// Mitsubishi GX Works2 project: ZhaoQing_OCV_1_9   PLC: Q06UDEH

TYPE ConveyorIO : STRUCT
  xCWPresent : BOOL;  (* 正转检测有无传感器 *)
  xCCWPresent : BOOL;  (* 反转检测有无传感器 *)
  xLoad : BOOL;  (* 上料请求 *)
  xUnload : BOOL;  (* 下料请求 *)
  xMotorCW : BOOL;  (* 电机正转 *)
  xMotorCCW : BOOL;  (* 电机反转 *)
  xEmpty : BOOL;  (* 线体状态为空 *)
  xNextRun : BOOL;  (* 下段线体运行 *)
  xUnloadCCW : BOOL;  (* 下料为反转 *)
  xloadCCW : BOOL;  (* 上料为反转 *)
  xForward : BOOL;  (* 正转手动 *)
  xBackward : BOOL;  (* 反转手动 *)
  xBusy : BOOL;  (* 工作中 *)
  xPutInto : BOOL;  (* 线体直接投入物料 *)
  xLoadAlarrm : BOOL;  (* 上料报警 *)
  xUnloadAlarm : BOOL;  (* 下料报警 *)
  iProductCategory : INT;  (* 产品种类 *)
  tLoadDelay : TIME;  (* 进入延时设置 *)
  tUnloadAlarmDelay : TIME;  (* 下料时间设置 *)
  xNotArriveAlarm : BOOL;  (* 未到达报警 *)
END_STRUCT END_TYPE

TYPE ShuttleCarIO : STRUCT
  xReady : BOOL;  (* 准备就绪 *)
  xForward : BOOL;  (* 正转 *)
  xBackward : BOOL;  (* 反转 *)
  iCurrentPos : INT;  (* 当前位置 *)
  iDestinationPos : INT;  (* 目标位置 *)
  xCW : BOOL;  (* 正转输出 *)
  xCCW : BOOL;  (* 反转输出 *)
  xBrake : BOOL;  (* 刹车 *)
  xHomeSwitch : BOOL;  (* 零位接近开关 *)
  xPosLimit : BOOL;  (* 正限位 *)
  xNegLimit : BOOL;  (* 负限位 *)
  xMDIExe : BOOL;  (* MDI开始 *)
  xMDIDone : BOOL;  (* MDI 完成 *)
  xPassLimit : BOOL;  (* 限位屏蔽 *)
  xPosLimitCatch : BOOL;  (* 正限位捕捉 *)
  xNegLimitCatch : BOOL;  (* 负限位捕捉 *)
  xHomeExe : BOOL;  (* 开始寻零 *)
  xHomeDone : BOOL;  (* 寻零完成 *)
  xHomeBusy : BOOL;  (* 寻零中 *)
  xHomeFailed : BOOL;  (* 寻零失败 *)
  xBusy : BOOL;  (* 工作中 *)
END_STRUCT END_TYPE

TYPE SwitchIO : STRUCT
  xLiftCylinderRetractDetect : BOOL;
  xLiftCylinderExtendDetect : BOOL;
  xLiftCylinderRetract : BOOL;
  xLiftCylinderExtend : BOOL;
  xEntryBarCylinderRetract : BOOL;
  xLiftCylinderExtendInit : BOOL;
  xEntryEnable : BOOL;
  xExitEnable : BOOL;
  xExitBarCylinderRetract : BOOL;
  xSwithEnable : BOOL;
  xLiftCylinderRetractButton : BOOL;
  xLiftCylinderExtendButton : BOOL;
  xEntryBarCylinderRetractButton : BOOL;
  xExitBarCylinderRetractButton : BOOL;
END_STRUCT END_TYPE

TYPE BarCylinderIO : STRUCT
  xBarCylinderButton : BOOL;  (* 阻挡气缸 *)
  xPresentSwitch : BOOL;  (* 行程开关 *)
  xBarCylinder : BOOL;  (* 阻挡气缸 *)
  xLoad : BOOL;  (* 上料 *)
  xEmpty : BOOL;  (* 为空指示 *)
  xNextRun : BOOL;  (* 下位设备开始运行 *)
  xUnload : BOOL;  (* 下料 *)
  xTransportMotorCWButton : BOOL;  (* 输送电机正转按钮 *)
  xTransportMotorCW : BOOL;  (* 输送电机正转 *)
  xTransportMotorCCWButton : BOOL;  (* 输送电机反转按钮 *)
  xTransportMotorCCW : BOOL;  (* 输送电机反转 *)
  iProductCategory : INT;  (* 产品种类 *)
  tLoadDelay : TIME;  (* 上料延时 *)
END_STRUCT END_TYPE

// global labels: Global1
VAR_GLOBAL
  g_xAuto AT M11 : BOOL;
  g_xManual : BOOL;
  g_xEStop AT X0BC : BOOL;
  g_xReset AT X0BE : BOOL;
  g_xStackLampRed AT Y2C1 : BOOL;
  g_xStackLampAmber AT Y2C3 : BOOL;
  g_xStackLampGreen AT Y2C2 : BOOL;
  g_xBuzzer AT Y2C4 : BOOL;
  g_xStop AT M2 : BOOL;
  g_xLocalAutoStart AT M1 : BOOL;
  g_xRemoteAutoStart AT M0 : BOOL;
  g_xRemoteAuto AT M10 : BOOL;
  g_iState AT D40 : INT;
  g_iLocalAutoStep : BOOL;
  g_xAlarm : BOOL;
END_VAR

// task Task_01 (event TRUE, interval 0, priority 31): POU, Start

FUNCTION_BLOCK Conveyor
VAR
  m_tLoadTimer : TIME;  (* 上料延时 *)
  m_tonNotArriveAlarm : TON;  (* 未到达报警计时 *)
  m_tonUnloadAlam : TON;  (* 下料报警定时器 *)
  m_tonLoadDelay : TON;  (* 上料延时 *)
  m_tUnloadTimer : TIME;  (* 下料计时器 *)
  iStep : INT;  (* 上料步骤 *)
  m_tNotArriveCurrentTime : TIME;  (* 未到达报警计时当前时间 *)
  m_xInitial : BOOL;  (* 初始化 *)
  m_xLoadDelayOut : BOOL;  (* 上料延时输出 *)
END_VAR
VAR_IN_OUT
  ConveyorMotor : ConveyorIO;  (* 输送线输入输出 *)
END_VAR
(*////////////////////////////////////////////////////////////////////////////////////////////////////////////
//传输线控制FB块，可控制单方向线体，双向旋转线体，支持双向上下料            
//线体初始化后为空的情况下输入xLoad信号即可进行上料动作，使用xLoadCCW信号可反方向上料
//增加了产品信息和产品种类的储存，当传输线为空和上料进行标志位为零的情况下清除产品信息和产品种类
//使用方式是在置位xLoad信号后，把产品信息和产品种类传入，等下料后自动清零
//线体不为空的情况下使用xUnload信号可进行下料动作，物料有无传感器的下降沿后出发计时器，延时断开传输线旋转
//单方向传输线体把xLoadCCW、xUnloadCCW设置为零，双向线体上料方向和下料反向的,方向固定的 把xUnloadCCW设置为1
//双方向线体双向都能上下料的要根据上料的方向来设置xLoadCCW,xUnloadCCW
//增加工作中信号xBusy当电机正转 显示为工作中
//增加上下料超时报警，xLoadAlarm，xUnloadAlarm，设定时间在LOAD_UNLOAD_TIME常量上，现在设置的为30秒
//增加xPutInto信号，用于直接投入的物料，检测开关感应到后，直接进入下料流程，上升沿有效
//离开延时改为变量 iLeaveDelay 默认为0 离开检测开关离输送线尾端比较远的线体需要根据情况设定100ms为单位
增加初始化标志位，增加进入延时时间，初始化为进入延时时间为0 ，离开延时时间为2S，通过外围接口可以更改
//修改信息  修改后请增加版本
12-17进行了优化，增加了未到达报警，当物料未传送到下一设备，就报未到达报警，使用xNextRun标志位制作，没有正常到达
第0步，不能跳转到第一步把标志位复位，即出现中断情况，2秒后报警 有问题

//YAO      V1.0
///////////////////////////////////////////////////////////////////////////////////////////////////////////
********************************************************)
IF NOT m_xInitial THEN
	ConveyorMotor.tLoadDelay:=T#0s;
	ConveyorMotor.tUnloadAlarmDelay:=T#30s;
	m_xInitial:=1;
END_IF;               (*初始化设置延时时间*)

CASE iStep OF
	0:
	ConveyorMotor.xMotorCW:=0;
	ConveyorMotor.xMotorCCW:=0;
    IF g_xAuto THEN          (*自动才进下一步*)
		IF (ConveyorMotor.xCWPresent OR ConveyorMotor.xCCWPresent)  THEN
			iStep:=3;
			ConveyorMotor.xEmpty:=0;(*检测到东西去3，复位empty*)
			ELSE
			iStep:=1;
			ConveyorMotor.xEmpty:=1;         (*没东西去1，置位empty*)
		END_IF;
	END_IF;
	1: 
	ConveyorMotor.xNextRun:=0;          (*复位NextRun*)
	IF ConveyorMotor.xLoad AND ConveyorMotor.xEmpty THEN	(*一般load接上一段的NextRun*)
		iStep:=2;                                             (*empty且有进料信号*)
	END_IF;
	2: 
	IF ConveyorMotor.xloadCCW THEN       (*如果正转为上料，则正转*)
		ConveyorMotor.xMotorCCW:=1; 
		ConveyorMotor.xMotorCW:=0;
	ELSE
	    ConveyorMotor.xMotorCW:=1;                (*反转为上料，则反转*)
		ConveyorMotor.xMotorCCW:=0;
	END_IF;
		m_tonLoadDelay(IN:= (ConveyorMotor.xCWPresent AND NOT ConveyorMotor.xloadCCW) 
		                                        OR (ConveyorMotor.xCCWPresent AND ConveyorMotor.xloadCCW) ,
		                               PT:= ConveyorMotor.tLoadDelay ,
		                               Q:= m_xLoadDelayOut ,
		                               ET:= m_tLoadTimer );
	    IF m_xLoadDelayOut THEN 	 
		    iStep:=3;                                             (*相应光电检测到东西，则去3*)
		END_IF;
	3:
	ConveyorMotor.xMotorCW:=0;
	ConveyorMotor.xMotorCCW:=0;
	ConveyorMotor.xEmpty:=0;          (*停转，且复位Empty，表示有料*)
	IF ConveyorMotor.xUnload THEN        (*停止运转，有Unload信号，则去4*)
		 iStep:=4;
	END_IF;
	4:	
	IF ConveyorMotor.xUnloadCCW THEN   (*正转为下料，则正转*)
		ConveyorMotor.xMotorCCW:=1;  
		ConveyorMotor.xMotorCW:=0;
		ELSE
	    ConveyorMotor.xMotorCW:=1;               (*反转为下料，则反转*)
		ConveyorMotor.xMotorCCW:=0;
	END_IF;
	ConveyorMotor.xNextRun:=1;         (*置位NextRun*)
	IF NOT ConveyorMotor.xUnload THEN       (*Unload信号为0则去0*)(*一般Unload由下段的Empty控制，即下段有料，流程走完*)
		istep:=0;
	END_IF;
END_CASE;
IF LDP(TRUE,ConveyorMotor.xPutInto) THEN
	iStep:=0;
END_IF;

(*IF ConveyorMotor.xEmpty AND iStep<>2 THEN
	ConveyorMotor.iProductCategory:=0;
END_IF;*)
IF g_xEStop=0 OR g_xReset THEN
	iStep:=0;
END_IF;	
IF g_xReset THEN
	ConveyorMotor.xNextRun:=0; 
END_IF;
IF g_xManual THEN
	iStep:=0;
	IF ConveyorMotor.xForward 
		AND ConveyorMotor.xBackward=0 
		AND ConveyorMotor.xMotorCCW=0
		AND g_xEStop THEN
		ConveyorMotor.xMotorCW:=1;
		ConveyorMotor.xMotorCCW:=0;
		ELSE
		ConveyorMotor.xMotorCW:=0;
	END_IF;

	IF ConveyorMotor.xBackward 
		AND ConveyorMotor.xForward=0 
		AND ConveyorMotor.xMotorCW=0
		AND g_xEStop  THEN
		ConveyorMotor.xMotorCCW:=1;
		conveyormotor.xMotorCW:=0;
		ELSE
		ConveyorMotor.xMotorCCW:=0;
	END_IF;
END_IF;
IF ConveyorMotor.xMotorCCW        
	OR ConveyorMotor.xMotorCW THEN  
	ConveyorMotor.xBusy:=1;
	ELSE
	ConveyorMotor.xBusy:=0;
END_IF;
m_tonNotArriveAlarm(IN:= iStep=0 AND ConveyorMotor.xNextRun,PT:= T#2s,Q:= ConveyorMotor.xNotArriveAlarm ,ET:= m_tNotArriveCurrentTime );
m_tonUnloadAlam(IN:= iStep=4,PT:=ConveyorMotor.tUnloadAlarmDelay,Q:= ConveyorMotor.xUnloadAlarm,ET:= m_tUnloadTimer );
END_FUNCTION_BLOCK

PROGRAM POU
VAR
  Cylinder12309 : ShuttleCar;
  CylinderIO12309 : ShuttleCarIO;
  ConveyorIO12114 : ConveyorIO;
  Conveyor12114 : Conveyor;
  Conveyor12115 : Conveyor;
  ConveyorIO12115 : ConveyorIO;
  Switch12312 : Switch;
  SwitchIO12312 : SwitchIO;
  Conveyor12123 : Conveyor;
  ConveyorIO12123 : ConveyorIO;
  Conveyor12124 : Conveyor;
  ConveyorIO12124 : ConveyorIO;
  Conveyor12125 : Conveyor;
  ConveyorIO12125 : ConveyorIO;
  Switch12203 : Switch;
  SwitchIO12203 : SwitchIO;
  Conveyor12142 : Conveyor;
  ConveyorIO12142 : ConveyorIO;
  Bar12326 : BarCylinder;
  BarIO12326 : BarCylinderIO;
  Conveyor12116 : Conveyor;
  ConveyorIO12116 : ConveyorIO;
  Cylinder12308 : ShuttleCar;
  CylinderIO12308 : ShuttleCarIO;
  Conveyor12111 : Conveyor;
  ConveyorIO12111 : ConveyorIO;
  Conveyor12112 : Conveyor;
  ConveyorIO12112 : ConveyorIO;
  Switch12311 : Switch;
  SwitchIO12311 : SwitchIO;
  Conveyor12113 : Conveyor;
  ConveyorIO12113 : ConveyorIO;
  Conveyor12120 : Conveyor;
  ConveyorIO12120 : ConveyorIO;
  Conveyor12121 : Conveyor;
  ConveyorIO12121 : ConveyorIO;
  Conveyor12122 : Conveyor;
  ConveyorIO12122 : ConveyorIO;
  Cylinder12307 : ShuttleCar;
  CylinderIO12307 : ShuttleCarIO;
  Conveyor12108 : Conveyor;
  ConveyorIO12108 : ConveyorIO;
  Conveyor12109 : Conveyor;
  ConveyorIO12109 : ConveyorIO;
  Switch12310 : Switch;
  SwitchIO12310 : SwitchIO;
  Conveyor12110 : Conveyor;
  ConveyorIO12110 : ConveyorIO;
  Conveyor12117 : Conveyor;
  ConveyorIO12117 : ConveyorIO;
  Conveyor12118 : Conveyor;
  ConveyorIO12118 : ConveyorIO;
  Conveyor12119 : Conveyor;
  ConveyorIO12119 : ConveyorIO;
  Conveyor12203 : Conveyor;
  ConveyorIO12203 : ConveyorIO;
  Conveyor12143 : Conveyor;
  ConveyorIO12143 : ConveyorIO;
  Switch12330 : Switch;
  ConveyorIO12144 : ConveyorIO;
  SwitchIO12330 : SwitchIO;
  Switch12333 : Switch;  (* OCV2顶升移载 *)
  ConveyorIO12333 : ConveyorIO;  (* OCV2顶升移载进入线体 *)
  ConveyorIO12152 : ConveyorIO;  (* OCV2顶升移载离开线体 *)
  SwitchIO12333 : SwitchIO;  (* OCV2顶升移载 *)
  m_xTS1ExportPermit : BOOL;  (* OCV2顶升移载 *)
  m_xConveyor12114Export : BOOL;  (* 12114线体输出 *)
  ConveyorIO12146 : ConveyorIO;
  m_xTS2ExportPermit : BOOL;
END_VAR
(*1巷道出库线体*)
Cylinder12309(ShuttleCarInOut:=CylinderIO12309);
ShuttleCarCurrentPosition( X43 OR X44 ,X44 ,X43, FALSE, CylinderIO12309.iCurrentPos );
CylinderIO12309.xReady:=TRUE;
CylinderIO12309.xForward:=M30;
CylinderIO12309.xBackward:=M31;
CylinderIO12309.xPosLimit:=1;
CylinderIO12309.xNegLimit:=1;
Y23D:=CylinderIO12309.xCW;
Y23C:=CylinderIO12309.xCCW;

Conveyor12114(ConveyorMotor:=ConveyorIO12114);
ConveyorIO12114.xForward:=M32;
ConveyorIO12114.xCWPresent:=X45;
Y23E:=ConveyorIO12114.xMotorCW;

Conveyor12115(ConveyorMotor:=ConveyorIO12115);
ConveyorIO12115.xForward:=M33;
ConveyorIO12115.xCWPresent:=X46;
Y23F:=ConveyorIO12115.xMotorCW;

Switch12312(ConveyorEntryIO:=ConveyorIO12116 ,
                                                        ConveyorExitIO:=ConveyorIO12123 ,
                                                        SwitchIO:=SwitchIO12312 );
SwitchIO12312.xLiftCylinderExtendButton:=M34;
SwitchIO12312.xLiftCylinderRetractButton:=M35;
Y242:=SwitchIO12312.xLiftCylinderExtend;
Y241:=SwitchIO12312.xLiftCylinderRetract;
SwitchIO12312.xLiftCylinderExtendDetect:=X4B;
SwitchIO12312.xLiftCylinderRetractDetect:=X4C;
ConveyorIO12116.xForward:=M36;
ConveyorIO12116.xCWPresent:=X49 OR X4A;
Y240:=ConveyorIO12116.xMotorCW;
ConveyorIO12123.xForward:=M37;
ConveyorIO12123.xCWPresent:=X49 OR X4A;
Y243:=ConveyorIO12123.xMotorCW;

Conveyor12124(ConveyorMotor:=ConveyorIO12124);
ConveyorIO12124.xForward:=M38;
ConveyorIO12124.xCWPresent:=X4D;
Y244:=conveyorIO12124.xMotorCW;

Conveyor12125(ConveyorMotor:=ConveyorIO12125);
ConveyorIO12125.xForward:=M39;
ConveyorIO12125.xCWPresent:=X4E;
Y245:=conveyorIO12125.xMotorCW;

(*2巷道出库线体*)
Cylinder12308(ShuttleCarInOut:=CylinderIO12308);
ShuttleCarCurrentPosition( X35 OR X36 ,X36 ,X35, FALSE, CylinderIO12308.iCurrentPos );
CylinderIO12308.xReady:=TRUE;
CylinderIO12308.xForward:=M40;
CylinderIO12308.xBackward:=M41;
CylinderIO12308.xPosLimit:=1;
CylinderIO12308.xNegLimit:=1;
Y235:=CylinderIO12308.xCW;
Y236:=CylinderIO12308.xCCW;

Conveyor12111(ConveyorMotor:=ConveyorIO12111);
ConveyorIO12111.xForward:=M42;
ConveyorIO12111.xCWPresent:=X37;
Y237:=ConveyorIO12111.xMotorCW;

Conveyor12112(ConveyorMotor:=ConveyorIO12112);
ConveyorIO12112.xForward:=M43;
ConveyorIO12112.xCWPresent:=X38;
Y238:=ConveyorIO12112.xMotorCW;

Switch12311(ConveyorEntryIO:=ConveyorIO12113 ,
                                                        ConveyorExitIO:=ConveyorIO12120 ,
                                                        SwitchIO:=SwitchIO12311 );
SwitchIO12311.xLiftCylinderExtendButton:=M44;
SwitchIO12311.xLiftCylinderRetractButton:=M45;
Y233:=SwitchIO12311.xLiftCylinderExtend;
Y232:=SwitchIO12311.xLiftCylinderRetract;
SwitchIO12311.xLiftCylinderExtendDetect:=X3D;
SwitchIO12311.xLiftCylinderRetractDetect:=X3E;
ConveyorIO12113.xForward:=M46;
ConveyorIO12113.xCWPresent:=X3B OR X3C;
Y239:=ConveyorIO12113.xMotorCW;
ConveyorIO12120.xForward:=M47;
ConveyorIO12120.xCWPresent:=X3B OR X3C;
Y234:=ConveyorIO12120.xMotorCW;

Conveyor12121(ConveyorMotor:=ConveyorIO12121);
ConveyorIO12121.xForward:=M48;
ConveyorIO12121.xCWPresent:=X3F;
Y23A:=conveyorIO12121.xMotorCW;

Conveyor12122(ConveyorMotor:=ConveyorIO12122);
ConveyorIO12122.xForward:=M49;
ConveyorIO12122.xCWPresent:=X40;
Y23B:=conveyorIO12122.xMotorCW;

(*3巷道出库线体*)
Cylinder12307(ShuttleCarInOut:=CylinderIO12307);
ShuttleCarCurrentPosition( X27 OR X28 ,X28 ,X27, FALSE, CylinderIO12307.iCurrentPos );
CylinderIO12307.xReady:=TRUE;
CylinderIO12307.xForward:=M50;
CylinderIO12307.xBackward:=M51;
CylinderIO12307.xPosLimit:=1;
CylinderIO12307.xNegLimit:=1;
Y228:=CylinderIO12307.xCW;
Y229:=CylinderIO12307.xCCW;

Conveyor12108(ConveyorMotor:=ConveyorIO12108);
ConveyorIO12108.xForward:=M52;
ConveyorIO12108.xCWPresent:=X26;
Y22A:=ConveyorIO12108.xMotorCW;

Conveyor12109(ConveyorMotor:=ConveyorIO12109);
ConveyorIO12109.xForward:=M53;
ConveyorIO12109.xCWPresent:=X25;
Y22B:=ConveyorIO12109.xMotorCW;

Switch12310(ConveyorEntryIO:=ConveyorIO12110 ,
                                                        ConveyorExitIO:=ConveyorIO12117 ,
                                                        SwitchIO:=SwitchIO12310 );
SwitchIO12310.xLiftCylinderExtendButton:=M54;
SwitchIO12310.xLiftCylinderRetractButton:=M55;
Y22D:=SwitchIO12310.xLiftCylinderExtend;
Y22E:=SwitchIO12310.xLiftCylinderRetract;
SwitchIO12310.xLiftCylinderExtendDetect:=X2D;
SwitchIO12310.xLiftCylinderRetractDetect:=X2E;
ConveyorIO12110.xForward:=M56;
ConveyorIO12110.xCWPresent:=X2F OR X30;
Y22C:=ConveyorIO12110.xMotorCW;
ConveyorIO12117.xForward:=M57;
ConveyorIO12117.xCWPresent:=X2F OR X30;
Y22F:=ConveyorIO12117.xMotorCW;

Conveyor12118(ConveyorMotor:=ConveyorIO12118);
ConveyorIO12118.xForward:=M58;
ConveyorIO12118.xCWPresent:=X31;
Y230:=conveyorIO12118.xMotorCW;

Conveyor12119(ConveyorMotor:=ConveyorIO12119);
ConveyorIO12119.xForward:=M59;
ConveyorIO12119.xCWPresent:=X32;
Y231:=conveyorIO12119.xMotorCW;
(*出库分流顶升移载*)
Switch12203(ConveyorEntryIO:=ConveyorIO12142 ,
                                                        ConveyorExitIO:=ConveyorIO12203 ,
                                                        SwitchIO:=SwitchIO12203);
SwitchIO12203.xLiftCylinderExtendButton:=M60;
SwitchIO12203.xLiftCylinderRetractButton:=M61;
SwitchIO12203.xExitBarCylinderRetractButton:=M64;
Y26B:=SwitchIO12203.xExitBarCylinderRetract;
Y269:=SwitchIO12203.xLiftCylinderExtend;
Y268:=SwitchIO12203.xLiftCylinderRetract;
SwitchIO12203.xLiftCylinderExtendDetect:=X88;
SwitchIO12203.xLiftCylinderRetractDetect:=X89;
ConveyorIO12142.xForward:=M62;
ConveyorIO12142.xCWPresent:=X86;
Y281:=ConveyorIO12142.xMotorCW;
ConveyorIO12142.tLoadDelay:=T#1s;
ConveyorIO12203.xForward:=M63;
ConveyorIO12203.xCWPresent:=X86;
Y26A:=ConveyorIO12203.xMotorCW;
SwitchIO12203.xLiftCylinderExtendInit:=0;

Bar12326(BarCylinderIO:=BarIO12326);
BarIO12326.tLoadDelay:=T#2s;
BarIO12326.xBarCylinderButton:=M64;
BarIO12326.xPresentSwitch:=X94;
BarIO12326.xTransportMotorCWButton:=M65;
Y26E:= BarIO12326.xTransportMotorCW;
Y26C:=BarIO12326.xBarCylinder;

Conveyor12143(ConveyorMotor:=ConveyorIO12143);
ConveyorIO12143.xForward:=M66;
ConveyorIO12143.xCWPresent:=XA2;
Y282:=ConveyorIO12143.xMotorCW;
(*OCV1顶升移载*)
Switch12330(ConveyorEntryIO:=ConveyorIO12144 ,
                                                        ConveyorExitIO:=ConveyorIO12146 ,
                                                        SwitchIO:=SwitchIO12330);
SwitchIO12330.xLiftCylinderExtendButton:=M67;
SwitchIO12330.xLiftCylinderRetractButton:=M68;
SwitchIO12330.xExitBarCylinderRetractButton:=M69;
Y286:=SwitchIO12330.xExitBarCylinderRetract;
Y284:=SwitchIO12330.xLiftCylinderExtend;
Y285:=SwitchIO12330.xLiftCylinderRetract;
SwitchIO12330.xLiftCylinderExtendDetect:=XA5;
SwitchIO12330.xLiftCylinderRetractDetect:=XA6;
ConveyorIO12144.xForward:=M70;
ConveyorIO12144.xCWPresent:=XA7;
Y283:=ConveyorIO12144.xMotorCW;
ConveyorIO12146.xForward:=M71;
ConveyorIO12146.xCWPresent:=XA7;
Y280:=ConveyorIO12146.xMotorCW;

(*OCV2顶升移载*)
Switch12333(ConveyorEntryIO:=ConveyorIO12333 ,
                                                        ConveyorExitIO:=ConveyorIO12152 ,
                                                        SwitchIO:=SwitchIO12333);
SwitchIO12333.xLiftCylinderExtendButton:=M72;
SwitchIO12333.xLiftCylinderRetractButton:=M73;
SwitchIO12333.xEntryBarCylinderRetractButton:=M74;
Y287:=SwitchIO12333.xEntryBarCylinderRetract;
Y289:=SwitchIO12333.xLiftCylinderExtend;
Y28A:=SwitchIO12333.xLiftCylinderRetract;
SwitchIO12333.xLiftCylinderExtendDetect:=XAC;
SwitchIO12333.xLiftCylinderRetractDetect:=XAD;
ConveyorIO12333.xForward:=M75;
ConveyorIO12333.xCWPresent:=XAB;
Y288:=ConveyorIO12333.xMotorCW;
ConveyorIO12333.tLoadDelay:=T#2s;
ConveyorIO12152.xForward:=M76;
ConveyorIO12152.xCWPresent:=XAB;
(*Y28B:=ConveyorIO12152.xMotorCW;*)
IF g_xManual THEN
	D3165:=0;
END_IF;
IF g_xAuto THEN
	(*与上位机接口程序
	"C1库出口(产品出库)
2014
出库完成状态	2165	"1：复位2：出库完成
出口状态	3165	"1:禁止出库2:允许出库"
1线堆积状态	3166	"1：正常2:堆积 "
2线堆积状态	3167	"1：正常2:堆积 "
3线堆积状态	3168	"1：正常2:堆积 "
    (**************************)
    IF NOT X41 AND NOT X42 AND CylinderIO12309.iCurrentPos=2 THEN
    	D3165:=2;
    ELSE
    	D3165:=1;
    END_IF;
   IF D2165=2 THEN
   		m_xTS1ExportPermit:=1;
   ELSE
   		m_xTS1ExportPermit:=0;
   END_IF;
   (**************************)
    (**************2巷道出库************) 
	IF NOT X33 
		AND NOT X34 
		AND ConveyorIO12111.xEmpty 
		AND ConveyorIO12112.xEmpty 
		AND NOT ConveyorIO12111.xBusy 
		AND NOT ConveyorIO12112.xBusy THEN
		CylinderIO12308.xMDIExe:=1;
		CylinderIO12308.iDestinationPos:=2;
	END_IF;
	IF m_xTS2ExportPermit=1 AND  X33 AND X34 THEN
		CylinderIO12308.xMDIExe:=1;
		CylinderIO12308.iDestinationPos:=1;
	END_IF;
	
	IF CylinderIO12308.iCurrentPos=1 AND X33 THEN
		ConveyorIO12111.xLoad:=1;
	ELSE
		ConveyorIO12111.xLoad:=0;
	END_IF;
	IF CylinderIO12308.iCurrentPos=1 AND X34 THEN
		ConveyorIO12112.xLoad:=1;
	ELSE
		ConveyorIO12112.xLoad:=0;	
	END_IF;	
	SwitchIO12311.xEntryEnable:=(ConveyorIO12111.xNextRun OR ConveyorIO12112.xNextRun) AND ConveyorIO12119.xEmpty ;
    ConveyorIO12111.xUnload:=ConveyorIO12113.xEmpty AND ConveyorIO12120.xEmpty AND NOT ConveyorIO12120.xBusy;
    SwitchIO12311.xSwithEnable:=1;
    IF LDP(TRUE,SwitchIO12311.xEntryEnable) THEN
  	  SwitchIO12311.xLiftCylinderExtendInit:=1;
    END_IF;
    SwitchIO12311.xExitEnable:=ConveyorIo12121.xEmpty;
    IF ConveyorIO12111.xEmpty AND conveyorIO12113.xEmpty AND NOT ConveyorIO12111.xBusy THEN
    	ConveyorIO12112.xUnload:=ConveyorIO12113.xEmpty AND ConveyorIO12120.xEmpty AND NOT ConveyorIO12120.xBusy;
    ELSE
    	ConveyorIO12112.xUnload:=0;
    END_IF;
    ConveyorIO12121.xLoad:=ConveyorIO12120 .xNextRun;
    ConveyorIO12121.xUnload:=ConveyorIO12122.xEmpty;
    ConveyorIO12122.xLoad:=ConveyorIO12121.xNextRun;
    IF LDP(TRUE,ConveyorIO12122.xEmpty=0) THEN
    	SwitchIO12312.xLiftCylinderExtendInit:=0;
    END_IF;
    ConveyorIO12122.xUnload:=ConveyorIO12123.xEmpty;
    ConveyorIO12123.xLoad:=ConveyorIO12122.xNextRun;
  (**************1巷道出库************) 
	IF NOT X41 
		AND NOT X42 
		AND ConveyorIO12114.xEmpty 
		AND ConveyorIO12115.xEmpty 
		AND NOT ConveyorIO12114.xBusy
		AND NOT ConveyorIO12115.xBusy THEN
		CylinderIO12309.xMDIExe:=1;
		CylinderIO12309.iDestinationPos:=2;
	END_IF;
	IF m_xTS1ExportPermit=1 AND  X41 AND X42 THEN
		CylinderIO12309.xMDIExe:=1;
		CylinderIO12309.iDestinationPos:=1;
	END_IF;
	
	IF CylinderIO12309.iCurrentPos=1 AND X41 THEN
		ConveyorIO12114.xLoad:=1;
	ELSE
		ConveyorIO12114.xLoad:=0;
	END_IF;
	IF CylinderIO12309.iCurrentPos=1  AND X42 THEN
		ConveyorIO12115.xLoad:=1;
	ELSE
		ConveyorIO12115.xLoad:=0;	
	END_IF;
	SwitchIO12312.xEntryEnable:=(ConveyorIO12114.xNextRun OR ConveyorIO12115.xNextRun) AND ConveyorIO12122.xEmpty ;
    ConveyorIO12114.xUnload:=ConveyorIO12116.xEmpty AND ConveyorIO12123.xEmpty AND NOT ConveyorIO12123.xBusy;
    SwitchIO12312.xSwithEnable:=1;
    IF ldp(TRUE,SwitchIO12312.xEntryEnable) THEN
  	  SwitchIO12312.xLiftCylinderExtendInit:=1;
    END_IF;
    SwitchIO12312.xExitEnable:=ConveyorIo12124.xEmpty;
    IF ConveyorIO12114.xEmpty AND conveyorIO12116.xEmpty AND NOT ConveyorIO12114.xBusy THEN
    	ConveyorIO12115.xUnload:=ConveyorIO12116.xEmpty AND ConveyorIO12123.xEmpty AND NOT ConveyorIO12123.xBusy;
    ELSE
    	ConveyorIO12115.xUnload:=0;
    END_IF;
    (*******************************************************************)
    ConveyorIO12124.xLoad:=ConveyorIO12123 .xNextRun;
    ConveyorIO12124.xUnload:=ConveyorIO12125.xEmpty;
    ConveyorIO12125.xLoad:=ConveyorIO12124.xNextRun;
     ConveyorIO12125.xUnload:=ConveyorIO12142.xEmpty;
    SwitchIO12203.xEntryEnable:=  ConveyorIO12125.xNextRun;
    SwitchIO12203.xSwithEnable:=0;
    SwitchIO12203.xExitEnable:=ConveyorIO12143.xEmpty;
    ConveyorIO12143.xLoad:=ConveyorIO12142.xNextRun;
    ConveyorIO12143.xUnload:=ConveyorIO12333.xEmpty;
    SwitchIO12333.xEntryEnable:=ConveyorIO12143.xNextRun;
	SwitchIO12333.xSwithEnable:=1;
	SwitchIO12333.xExitEnable:=NOT XAE;
END_IF;
END_PROGRAM

FUNCTION_BLOCK PriorityFB
VAR_INPUT
  xCondition1 : BOOL;  (* 条件1 *)
  xCondition2 : BOOL;  (* 条件2 *)
  xCondition3 : BOOL;  (* 条件3 *)
  xCondition4 : BOOL;  (* 条件4 *)
  xCondition5 : BOOL;  (* 条件5 *)
  xTaskComplete : BOOL;  (* 任务完成 *)
  xReset : BOOL;  (* 复位 *)
END_VAR
VAR
  xOccupy : BOOL;  (* 占用 *)
END_VAR
VAR_OUTPUT
  iPriority : INT;  (* 输出任务号 *)
END_VAR
VAR
  m_tonConditionDelay : TON;
  m_xConditionDelay : BOOL;
  m_tConditionCurrentTime : TIME;
END_VAR
(*我在reset那里加了Occupy的复位
任务为0时，Occupy也会自动复位
*)
IF NOT xCondition1 
	AND NOT xCondition2
	AND NOT xCondition3
	AND NOT xCondition4
	AND NOT xCondition5
	AND NOT xOccupy  THEN
	iPriority:=0;
END_IF;
IF LDP(TRUE, xTaskComplete) THEN
	xOccupy:=0;
	iPriority:=0;
END_IF;
m_tonConditionDelay(IN:= (xCondition1
                                                     OR  xCondition2
                                                     OR  xCondition3
                                                     OR  xCondition4
                                                     OR xCondition5)
                                                     AND iPriority=0,
                                                     PT:= T#1s,
                                                     Q:= m_xConditionDelay ,
                                                     ET:= m_tConditionCurrentTime );
IF xCondition1 AND NOT xOccupy AND m_xConditionDelay THEN
	iPriority:=1;
	xOccupy:=1;
END_IF;
IF xCondition2 AND NOT xOccupy AND m_xConditionDelay  THEN
	iPriority:=2;
	xOccupy:=1;
END_IF;
IF xCondition3 AND NOT xOccupy AND m_xConditionDelay  THEN
	iPriority:=3;
	xOccupy:=1;
END_IF;
IF xCondition4 AND NOT xOccupy AND m_xConditionDelay  THEN
	iPriority:=4;
	xOccupy:=1;
END_IF;
IF xCondition5 AND NOT xOccupy AND m_xConditionDelay  THEN
	iPriority:=5;
	xOccupy:=1;
END_IF;

IF xReset THEN
	iPriority:=0;
	xOccupy:=0;
END_IF;
IF iPriority=0 THEN
	xOccupy:=0;
END_IF;
END_FUNCTION_BLOCK

FUNCTION_BLOCK ShuttleCar
VAR_IN_OUT
  ShuttleCarInOut : ShuttleCarIO;
END_VAR
VAR
  m_xBrakeDelay : BOOL;  (* 刹车延时标志位 *)
  diCurrentPosRetain : DINT;
  m_tonBrakeDelay : TON;  (* 延时 *)
  m_tBrakeDelay : TIME;
  m_xBrake : BOOL;
  m_tBrakeDelayCurrentTime : TIME;
END_VAR
(*******************************************************************
输送小车程序，可用于使用认址片控制位置的输送车程序，可用于控制提升机，
使用了限位捕捉程序防止小车惯性过大冲过限位后继续行走，捕捉程序采用反
转复位，这样设计有弊端可能反转复位后车的位置并没有回到限位以内,当两个
限位同时碰到的时候，会使运料小车进入死锁状态，通过xPassLimit来解开死锁，
可以在触摸屏中使用一个带权限的按钮来进行控制，配合ShuttleCarCurrentPos
函数来计算位置信息
增加自动开始后将当前位置置为零的信号防止设备停在两个位置开关的中间
修改信息  修改后请增加版本
YAO      V1.0
********************************************************************)

ShuttleCarInOut.xPosLimitCatch:=LDF(TRUE,ShuttleCarInOut.xPosLimit) OR ShuttleCarInOut.xPosLimitCatch;
IF ShuttleCarInOut.xCCW THEN  
	ShuttleCarInOut.xPosLimitCatch:=0;
END_IF;

ShuttleCarInOut.xNegLimitCatch:=LDF(TRUE,ShuttleCarInOut.xNegLimit) OR ShuttleCarInOut.xNegLimitCatch;
IF ShuttleCarInOut.xCW THEN   
	ShuttleCarInOut.xNegLimitCatch:=0;  
END_IF;
IF ShuttleCarInOut.xPassLimit OR
	(ShuttleCarInOut.xNegLimitCatch 
	AND ShuttleCarInOut.xPosLimitCatch)  THEN  
	ShuttleCarInOut.xNegLimitCatch:=0; 
	ShuttleCarInOut.xPosLimitCatch:=0;
END_IF;

IF ShuttleCarInOut.xReady THEN	
    IF g_xManual THEN  
	    IF ShuttleCarInOut.xForward 
			AND ShuttleCarInOut.xBackward=0 
			AND ShuttleCarInOut.xCCW=0 
			AND ShuttleCarInOut.xPosLimitCatch=0 
			AND g_xEStop THEN
		    ShuttleCarInOut.xCW:=1;
		    ELSE
		    ShuttleCarInOut.xCW:=0;
	    END_IF;
	    IF ShuttleCarInOut.xBackward 
			AND ShuttleCarInOut.xForward=0 
			AND ShuttleCarInOut.xCW=0 
			AND ShuttleCarInOut.xNegLimitCatch=0 
			AND G_xEStop THEN  
		    ShuttleCarInOut.xCCW:=1;
		    ELSE
		    ShuttleCarInOut.xCCW:=0;
	    END_IF;
    END_IF;
  IF g_xAuto AND g_xEStop THEN  
	  IF ShuttleCarInOut.xMDIExe AND ShuttleCarInOut.iDestinationPos<>0 THEN
	
	    IF ShuttleCarInOut.iCurrentPos<ShuttleCarInOut.iDestinationPos AND ShuttleCarInOut.xPosLimitCatch=0 THEN
			ShuttleCarInOut.xCW:=1;
			ShuttleCarInOut.xCCW:=0;
			ShuttleCarInOut.xMDIDone:=0;
		END_IF;

		IF ShuttleCarInOut.iCurrentPos>ShuttleCarInOut.iDestinationPos AND ShuttleCarInOut.xNegLimitCatch=0 THEN
			ShuttleCarInOut.xCCW:=1;
			ShuttleCarInOut.xCW:=0;
			ShuttleCarInOut.xMDIDone:=0;
		END_IF;
	
		IF ShuttleCarInOut.iCurrentPos=ShuttleCarInOut.iDestinationPos THEN
			ShuttleCarInOut.xCW:=0;
			ShuttleCarInOut.xCCW:=0;
			ShuttleCarInOut.xMDIDone:=1;
			ELSE
			ShuttleCarInOut.xMDIDone:=0;
		END_IF;

		IF ShuttleCarInOut.xPosLimitCatch THEN
			ShuttleCarInOut.xCW:=0;
			ShuttleCarInOut.xMDIDone:=0;
		END_IF;

		IF ShuttleCarInOut.xNegLimitCatch THEN
			ShuttleCarInOut.xCCW:=0;
			ShuttleCarInOut.xMDIDone:=0;
		END_IF;
		ELSE
		ShuttleCarInOut.xCW:=0;
		ShuttleCarInOut.xCCW:=0;
		ShuttleCarInOut.xMDIDone:=0;
	  END_IF;
	END_IF;
	ELSE
		ShuttleCarInOut.xCW:=0;
		ShuttleCarInOut.xCCW:=0;	
END_IF;
m_tonBrakeDelay(IN:=m_xBrakeDelay ,PT:= T#100ms,Q:=m_xBrake ,ET:= m_tBrakeDelayCurrentTime);
IF (ShuttleCarInOut.xCW OR ShuttleCarInOut.xCCW) AND ShuttleCarInOut.xReady=1 THEN
	ShuttleCarInOut.xBrake:=m_xBrake;
	m_xBrakeDelay:=1;
	ELSE
	ShuttleCarInOut.xBrake:=0;
	m_xBrakeDelay:=0;
END_IF;

IF g_xEStop =0 THEN
	ShuttleCarInOut.xCW :=0;
	ShuttleCarInOut.xCCW:=0;
END_IF;

(*IF SM402 THEN 
	ShuttleCarInOut.diCurrentPos:=diCurrentPosRetain;
	ELSE
	diCurrentPosRetain:=ShuttleCarInOut.diCurrentPos;
END_IF;*)
(*自动上电后把当前位置清零，防止穿梭车不在开关位置*)
IF LDP(TRUE,g_xAuto) THEN
	ShuttleCarInOut.iCurrentPos:=0;
END_IF;
IF ShuttleCarInOut.xCW OR ShuttleCarInOut.xCCW THEN
	ShuttleCarInOut.xBusy:=1;
	ELSE
	ShuttleCarInout.xBusy:=0;
END_IF;
END_FUNCTION_BLOCK

FUNCTION ShuttleCarCurrentPosition
VAR_INPUT
  xPosition1 : BOOL;
  xPosition2 : BOOL;
  xPosition3 : BOOL;
END_VAR
(************************************
计算输送车当前位置的函数
**************************************)
IF xPosition1 THEN
	ShuttleCarCurrentPosition:=1;
END_IF;
IF xPosition2 THEN
	ShuttleCarCurrentPosition:=2;
END_IF;
IF xPosition3 THEN
	ShuttleCarCurrentPosition:=3;
END_IF;
END_FUNCTION

FUNCTION ShuttleCarVelocityEncoder
VAR_INPUT
  iDestinationPos : INT;  (* 目标位置 *)
  iCurrentPos : INT;  (* 当前位置 *)
  xEnable : BOOL;  (* 使能 *)
END_VAR
IF xEnable THEN
	IF ABS(iCurrentPos-iDestinationPos)<300  THEN
		ShuttleCarVelocityEncoder:=0;
	ELSE
		ShuttleCarVelocityEncoder:=1;
	END_IF;
ELSE
	ShuttleCarVelocityEncoder:=0;
END_IF;
END_FUNCTION

FUNCTION_BLOCK ShuttleCarVelocityFB
VAR_INPUT
  xEnable : BOOL;  (* 使能 *)
  xMotorCW : BOOL;  (* 电机正转 *)
  xMotorCCW : BOOL;  (* 电机反转 *)
  xPosition1Switch : BOOL;  (* 位置1开关 *)
  xDecelerationSwitch : BOOL;  (* 减速开关 *)
  xPosition2Switch : BOOL;  (* 位置2开关 *)
END_VAR
VAR
  iFloor : INT;  (* 层数 *)
END_VAR
VAR_OUTPUT
  xHighSpeed : BOOL;
END_VAR
IF xEnable THEN
	(*电机旋转，并且在位置开关上的时候触发加速*)
	IF( LDP(TRUE,xMotorCW) AND xPosition1Switch ) OR (  LDP(TRUE,xMotorCCW) AND xPosition2Switch) THEN
		xHighSpeed:=1;
		iFloor:=0;
	END_IF;
	IF LDF(TRUE,xMotorCW) OR LDF(TRUE,xMotorCCW) THEN
		xHighSpeed:=0;
    END_IF;
	IF LDP(TRUE,xDecelerationSwitch) THEN
		iFloor:=iFloor+1;
	END_IF;
	IF iFloor=2 THEN
		xHighSpeed:=0;
		iFloor:=0;
	END_IF;
ELSE
    xHighSpeed:=0;
END_IF;
END_FUNCTION_BLOCK

PROGRAM Start
IF g_xReset THEN
	SM50:=1;
ELSE
	SM50:=0;
END_IF;
CASE g_iState OF
	0: 
		g_xManual:=1;
		g_xAuto:=0;	
		g_xStackLampAmber:=1;
		g_xStackLampGreen:=0;
		g_xRemoteAuto:=0;
	1:
		g_xManual:=0;
		g_xAuto:=1;
		g_xStackLampGreen:=1;
		g_xStackLampAmber:=0;
		g_xRemoteAuto:=0;
	2:	
        g_xRemoteAuto:=1;
        g_xStackLampGreen:=1;
        g_xStackLampAmber:=0;
        g_xAuto:=0;
		g_xManual:=0;
END_CASE;
IF g_xLocalAutoStart THEN  
	g_iState:=1;
END_IF;
IF g_xAlarm AND SM412 THEN
	g_xStackLampRed:=1;
	g_xBuzzer:=1;
ELSE
	g_xStackLampRed:=0;
	g_xBuzzer:=0;	
END_IF;
IF g_xStop OR g_xEStop=0 THEN 
	g_iState:=0;
END_IF;
IF g_xRemoteAutoStart THEN
	g_iState:=2;
END_IF;
END_PROGRAM

FUNCTION_BLOCK Switch
VAR_IN_OUT
  ConveyorEntryIO : ConveyorIO;
END_VAR
VAR
  ConveyorEntry : Conveyor;
END_VAR
VAR_IN_OUT
  ConveyorExitIO : ConveyorIO;
END_VAR
VAR
  m_tonLiftCylinderDelay : TON;  (* 顶升延时 *)
  m_xLiftCylinderDelay : BOOL;
  m_tLiftCylinderDelay : TIME;
  m_tonExitBarDelay : TON;  (* 退出阻挡器延时 *)
  m_tExitBarDelay : TIME;
  m_xExitBarDelay : BOOL;
END_VAR
VAR_IN_OUT
  SwitchIO : SwitchIO;
END_VAR
VAR
  iStep : INT;
  ConveyorExit : Conveyor;
  m_xInitial : BOOL;
END_VAR
(**************************************************
顶升移载模块，抽象为一条输入输线 ，一条输出输送线
一个进入阻挡器，一个放出阻挡器，和一个顶升气缸的控制
程序思路比较混乱，接口不清晰，需要整改
直接放行的时候有问题
switchEnable =0的时候   离开线体的PutInto有问题
12-17日   V1.0
***************************************************)
ConveyorEntry(ConveyorMotor:=ConveyorEntryIO);
ConveyorExit(ConveyorMotor:=ConveyorExitIO);

IF NOT m_xInitial THEN
	
	m_xInitial:=1;
END_IF;
IF g_xAuto THEN
	CASE iStep OF
		0:(*初始化*)
		ConveyorEntryIO.xLoad:=0;
		ConveyorEntryIO.xUnload:=0;
		ConveyorEntryIO.xPutInto:=0;
		ConveyorExitIO.xLoad:=0;
		ConveyorExitIo.xUnload:=0;
		ConveyorExitIO.xPutInto:=0;
		SwitchIO.xEntryBarCylinderRetract:=0;
		SwitchIO.xExitBarCylinderRetract:=0;
		IF SwitchIO.xLiftCylinderExtendInit THEN
			SwitchIO.xLiftCylinderExtend:=1;
			SwitchIO.xLiftCylinderRetract:=0;
		    IF SwitchIO.xLiftCylinderExtendDetect THEN
			    iStep:=1;
		     END_IF; 
		ELSE
			SwitchIO.xLiftCylinderExtend:=0;
			SwitchIO.xLiftCylinderRetract:=1;	
		    IF SwitchIO.xLiftCylinderRetractDetect THEN
			    iStep:=1;
		    END_IF;		
		END_IF;
		1:(*上料*)
        IF SwitchIO.xEntryEnable AND ConveyorEntryIO.xEmpty AND ConveyorExitIO.xEmpty THEN
        	SwitchIO.xEntryBarCylinderRetract:=1;
        	ConveyorEntryIO.xLoad:=1;
        END_IF;
        IF ConveyorEntryIO.xEmpty=0 THEN
        	SwitchIO.xEntryBarCylinderRetract:=0;
        	ConveyorEntryIO.xLoad:=0;
        	ConveyorExitIO.xPutInto:=1;
        END_IF;
        IF m_xLiftCylinderDelay AND  SwitchIO.xSwithEnable THEN
        	 iStep:=2;
        END_IF;
        IF SwitchIO.xSwithEnable=0 AND m_xLiftCylinderDelay  THEN
        	 iStep:=3;
        END_IF;
		2:(*顶升*)
			SwitchIO.xExitBarCylinderRetract:=0;
		    IF SwitchIO.xLiftCylinderExtendInit THEN
			    SwitchIO.xLiftCylinderExtend:=0;
			    SwitchIO.xLiftCylinderRetract:=1;
		    ELSE
			    SwitchIO.xLiftCylinderExtend:=1;
			    SwitchIO.xLiftCylinderRetract:=0;			
		   END_IF;

		  IF SwitchIO.xLiftCylinderExtendInit THEN
		  	IF SwitchIO.xLiftCylinderRetractDetect THEN
		  		iStep:=4;
		  	END_IF;
		  	ELSE
		  	IF SwitchIO.xLiftCylinderExtendDetect THEN
		      iStep:=4; 
		  	END_IF;
		  END_IF;
		  3:(*放行*)	
		  	SwitchIO.xExitBarCylinderRetract:=1;
		  	ConveyorExitIO.xPutInto:=0;
		  	iStep:=4;
		  4:(*下料*)
		  (*通过出料传输线下料*)
		  IF SwitchIO.xExitEnable  AND m_xExitBarDelay AND NOT SwitchIO.xExitBarCylinderRetract  THEN		  
		  	ConveyorExitIO.xUnload:=1;
		  ELSE
		  	ConveyorExitIO.xUnload:=0;
		  END_IF;	
		   (*通过进料传输线下料*)
		  IF SwitchIO.xExitEnable  AND m_xExitBarDelay  AND SwitchIO.xExitBarCylinderRetract THEN		  
		  	ConveyorEntryIO.xUnload:=1;
		  ELSE
		  	ConveyorEntryIO.xUnload:=0;
		  END_IF;			    	
		  IF (ConveyorExitIO.xEmpty OR ConveyorEntryIO.xEmpty) AND m_xExitBarDelay  THEN
		  	ConveyorExitIO.xPutInto:=1;
		  	ConveyorEntryIO.xPutInto:=1;
			iStep:=0; 
		  END_IF;
	END_CASE;
        m_tonLiftCylinderDelay(IN:=NOT ConveyorEntryIO.xEmpty AND iStep=1 ,PT:= T#1S ,Q:= m_xLiftCylinderDelay ,ET:=m_tLiftCylinderDelay );
 		m_tonExitBarDelay(IN:=iStep=4 ,PT:= T#1s ,Q:= m_xExitBarDelay ,ET:= m_tExitBarDelay);
END_IF;
IF g_xReset OR LDP(TRUE,SwitchIO.xLiftCylinderExtendInit) OR LDF(TRUE,SwitchIO.xLiftCylinderExtendInit) THEN
	iStep:=0;
END_IF;
IF g_xManual  THEN
	iStep:=0;
	ConveyorEntryIO.xLoad:=0;
    ConveyorEntryIO.xUnload:=0;
	ConveyorEntryIO.xPutInto:=0;
	ConveyorExitIO.xLoad:=0;
	ConveyorExitIo.xUnload:=0;
	ConveyorExitIO.xPutInto:=0;
	SwitchIO.xEntryBarCylinderRetract:=0;
	SwitchIO.xExitBarCylinderRetract:=0;
	IF SwitchIO.xEntryBarCylinderRetractButton THEN
		SwitchIO.xEntryBarCylinderRetract:=1;
	ELSE
		SwitchIO.xEntryBarCylinderRetract:=0;
	END_IF;
		IF SwitchIO.xExitBarCylinderRetractButton THEN
		SwitchIO.xExitBarCylinderRetract:=1;
	ELSE
		SwitchIO.xExitBarCylinderRetract:=0;
		END_IF;
		IF SwitchIO.xLiftCylinderExtendButton AND NOT SwitchIO.xLiftCylinderRetractButton THEN
			SwitchIO.xLiftCylinderExtend:=1;
			SwitchIO.xLiftCylinderRetract:=0;
		END_IF;
		IF NOT SwitchIO.xLiftCylinderExtendButton AND  SwitchIO.xLiftCylinderRetractButton THEN
			SwitchIO.xLiftCylinderExtend:=0;
			SwitchIO.xLiftCylinderRetract:=1;
		END_IF;		
	END_IF;
END_FUNCTION_BLOCK

FUNCTION_BLOCK BarCylinder
VAR_IN_OUT
  BarCylinderIO : BarCylinderIO;
END_VAR
VAR
  m_xInitial : BOOL;  (* 初始化 *)
  m_tonLoadDelay : TON;  (* 上料延时 *)
  m_xLoadDelay : BOOL;  (* 上料延时标志位 *)
  m_tLoadDelayCurrentTime : TIME;  (* 上料延时当前时间 *)
END_VAR
  (***********************************************************************
阻挡器模块，
由一个行程开关，一个阻挡器，一个倍速链输送电机组成
具有手动与自动模式
xEmpty显示当前为空料的状态
xUnload为卸料信号，连接下一设备的xEmpty信号
*************************************************************************)

IF NOT m_xInitial THEN
	BarCylinderIO.tLoadDelay:=T#5s;
	m_xInitial:=1;
END_IF;
IF g_xManual THEN    (*手动*)
	BarCylinderIO.xNextRun:=0;
	IF BarCylinderIO.xBarCylinderButton THEN
		BarCylinderIO.xBarCylinder:=1;
	ELSE
		BarCylinderIO.xBarCylinder:=0;
	END_IF;
	IF BarCylinderIO.xTransportMotorCWButton 
		AND NOT BarCylinderIO.xTransportMotorCCWButton 
		AND NOT BarCylinderIO.xTransportMotorCCW   THEN
		BarCylinderIO.xTransportMotorCW:=1;
	ELSE
		BarCylinderIO.xTransportMotorCW:=0;
	END_IF;
	IF BarCylinderIO.xTransportMotorCCWButton 
		AND NOT BarCylinderIO.xTransportMotorCWButton 
		AND NOT BarCylinderIO.xTransportMotorCW   THEN
		BarCylinderIO.xTransportMotorCCW:=1;
	ELSE
		BarCylinderIO.xTransportMotorCCW:=0;
	END_IF;
END_IF;
IF g_xAuto THEN(*自动*)
    IF BarCylinderIO.xUnload  AND NOT BarCylinderIO.xEmpty AND NOT BarCylinderIO.xNextRun THEN(*收到卸料命令，当阻挡器不为空时*)
    	BarCylinderIO.xBarCylinder:=1;
    	BarCylinderIO.xNextRun:=1;(*确保下料命令只执行一次，防止物料在输送过程中又有卸料命令导致多次卸料*)
    	BarCylinderIO.xTransportMotorCW:=1;
    END_IF;
    IF NOT  BarCylinderIO.xUnload  THEN
    	BarCylinderIO.xNextRun:=0;
    	BarCylinderIO.xBarCylinder:=0;
    END_IF;
    m_tonLoadDelay(IN:= BarCylinderIO.xPresentSwitch ,PT:= BarCylinderIO.tLoadDelay ,Q:= m_xLoadDelay,ET:= m_tLoadDelayCurrentTime );
    IF m_xLoadDelay OR  BarCylinderIO.xNextRun  THEN
    	BarCylinderIO.xEmpty:=0;
    ELSE
    	BarCylinderIO.xEmpty:=1;
    END_IF;
    (*如果为空，气缸顶起*)
   IF  BarCylinderIO.xEmpty  THEN
   	   BarCylinderIO.xBarCylinder:=0;
   END_IF;
   	IF BarCylinderIO.xLoad AND BarCylinderIO.xEmpty  THEN
		BarCylinderIO.xTransportMotorCW:=1;
   	END_IF;  
   	IF (BarCylinderIO.xLoad=0 OR BarCylinderIO.xEmpty=0)  AND (BarCylinderIO.xUnload=0 OR BarCylinderIO.xEmpty) THEN
   		BarCylinderIO.xTransportMotorCW:=0;
   	END_IF;
END_IF;  
IF BarCylinderIO.xEmpty AND BarCylinderIO.xLoad=0 THEN
	BarCylinderIO.iProductCategory:=0;
END_IF;

IF NOT g_xEStop THEN
	 BarCylinderIO.xTransportMotorCW:=0;
	 BarCylinderIO.xTransportMotorCCW:=0;
	 BarCylinderIO.xBarCylinder:=0;
END_IF;
END_FUNCTION_BLOCK
